// TIA Portal V19 program export: 1 tag tables, 0 data types, 0 data blocks, 1 code blocks (in call order from the OBs), 0 instance data blocks

VAR_GLOBAL   // PLC tag table "Default tag table"
   System_Byte AT %MB1 : Byte;
   FirstScan AT %M1.0 : Bool;
   DiagStatusUpdate AT %M1.1 : Bool;
   AlwaysTRUE AT %M1.2 : Bool;
   AlwaysFALSE AT %M1.3 : Bool;
   Clock_Byte AT %MB0 : Byte;
   Clock_10Hz AT %M0.0 : Bool;
   Clock_5Hz AT %M0.1 : Bool;
   "Clock_2.5Hz" AT %M0.2 : Bool;
   Clock_2Hz AT %M0.3 : Bool;
   "Clock_1.25Hz" AT %M0.4 : Bool;
   Clock_1Hz AT %M0.5 : Bool;
   "Clock_0.625Hz" AT %M0.6 : Bool;
   "Clock_0.5Hz" AT %M0.7 : Bool;
   "to 1500rh" AT %QB100 : Byte;
   "from 1500RH" AT %IB100 : Byte;
   "to 1500rh_right" AT %QB200 : Byte;
   "from 1500rh_right" AT %IB200 : Byte;
END_VAR

ORGANIZATION_BLOCK "Main"   // OB1, LAD, ProgramCycle
TITLE = "Main Program Sweep (Cycle)"
{ S7_Optimized_Access := 'TRUE' }
// stored: SetENOAutomatically false
   VAR_INPUT
      Initial_Call : Bool;   // Initial call of this OB
      Remanence : Bool;   // =True, if remanent data are available
   END_VAR
BEGIN

REGION Network 1
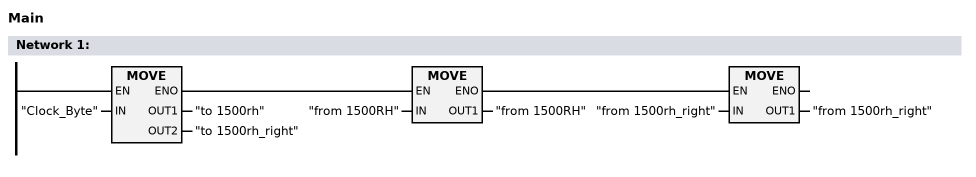
   RUNG wire#powerrail
      Move(in := "Clock_Byte", out1 => "to 1500rh", out2 => "to 1500rh_right")
      Move(in := "from 1500RH", out1 => "from 1500RH")
      Move(in := "from 1500rh_right", out1 => "from 1500rh_right")
   END_RUNG
   // the same network as SCL:
   "to 1500rh" := "Clock_Byte";
   "to 1500rh_right" := "Clock_Byte";
   "from 1500RH" := "from 1500RH";
   "from 1500rh_right" := "from 1500rh_right";
END_REGION
END_ORGANIZATION_BLOCK
